// TIA Portal V17 export
// export: Created 2025-03-13T10:29:52.3164471Z, ExportSetting WithDefaults, DisplayName Totally Integrated Automation Portal, DisplayVersion V17 Update 8, DisplayName TIA Portal Openness, DisplayVersion V17 Update 8, DisplayName TIA Portal Version Control Interface, DisplayVersion V17, DisplayName SINAMICS Startdrive Advanced, DisplayVersion V17 SP2, DisplayName SINAMICS Startdrive G110M, G120, G120C, G120D, G120P, G115D, DisplayVersion V17 SP2, DisplayName SINAMICS Startdrive G130, G150, S120, S150, SINAMICS MV, S210, DisplayVersion V17 SP2, DisplayName STEP 7 Professional, DisplayVersion V17 Update 8, DisplayName SINUMERIK ONE STEP 7 Toolbox, DisplayVersion V17 Update 12, DisplayName SINUMERIK 840D sl STEP 7 Toolbox, DisplayVersion V17 Update 12, DisplayName STEP 7 Safety, DisplayVersion V17 Update 6, DisplayName WinCC Advanced, DisplayVersion V17 Update 8
FUNCTION "FC7455_QUALITY_PART_COUNTER_CLADDING" : Void   // FC7455, LAD
{ S7_Optimized_Access := 'FALSE' }
AUTHOR : ETXETAR
NAME : GM-QC
VERSION : 1.0
// stored: AutoNumber false, IsIECCheckEnabled false, SetENOAutomatically false, UDAEnableTagReadback false
   VAR_TEMP
      VALUE_0 : Real;
      AUX_FAULT : Bool;
   END_VAR
   VAR CONSTANT
      FC_NUMBER : DInt := 7455;
   END_VAR
   VAR_TEMP   // added for the SCL form of the ladder/FBD networks
      _w1 : Bool;
      _w2 : Bool;
   END_VAR
BEGIN

REGION Network 1: PART COUNTER
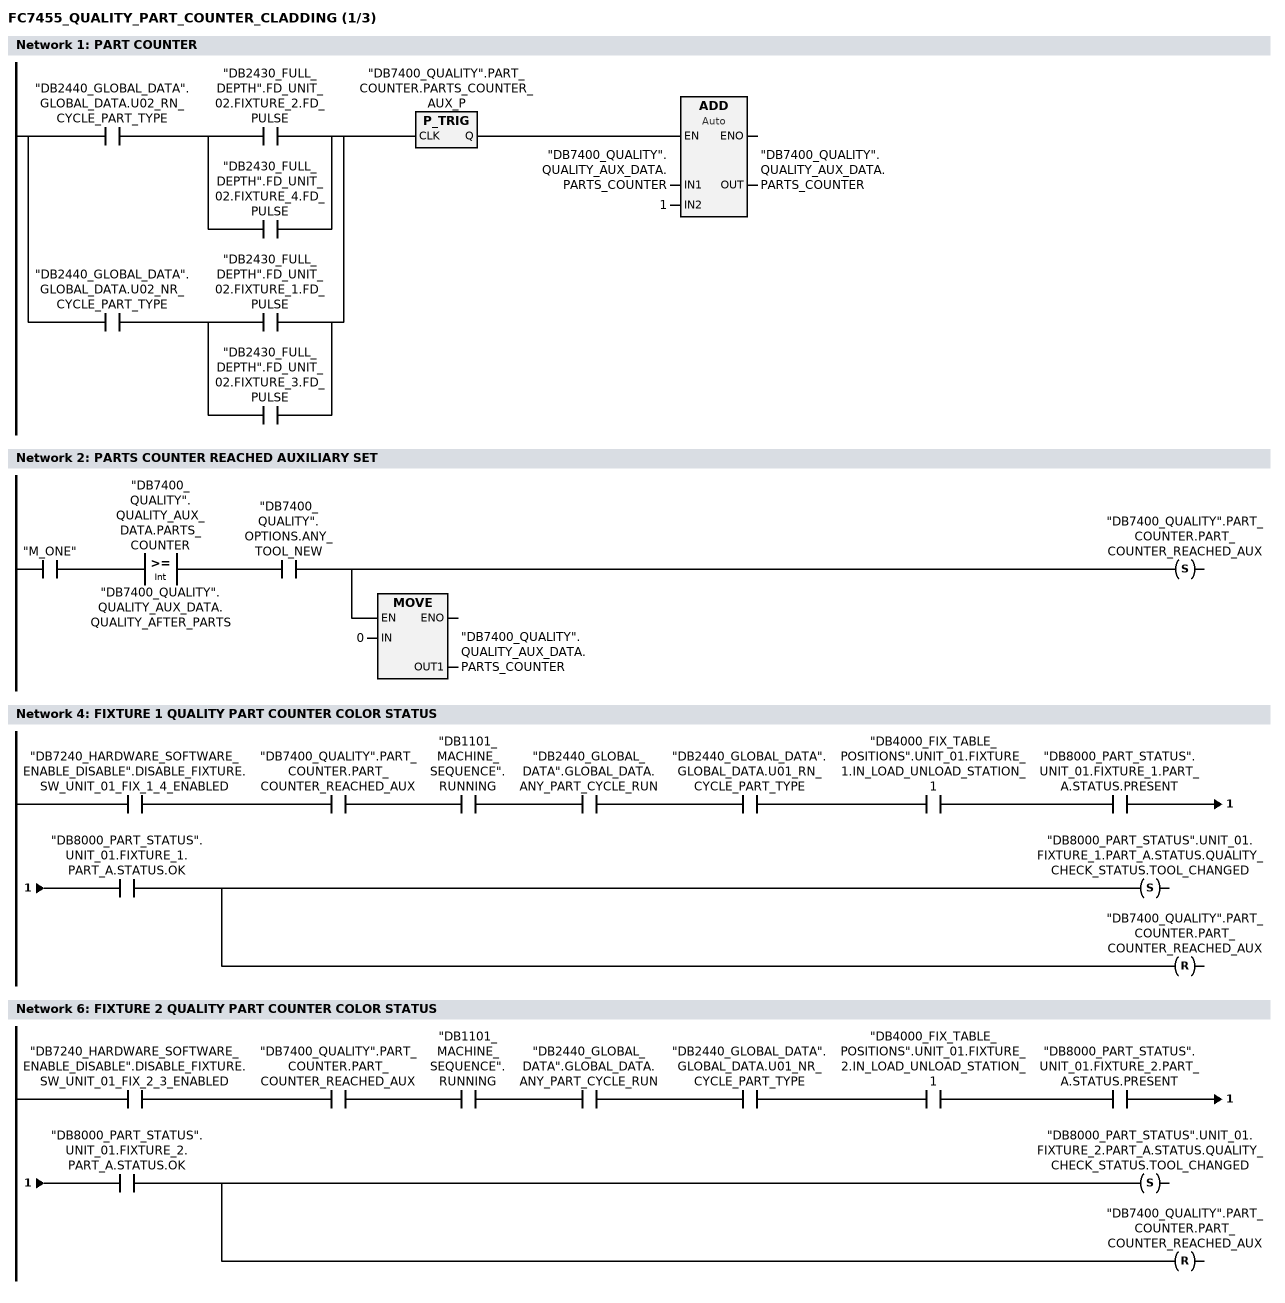
   RUNG wire#powerrail
      Contact( "DB2440_GLOBAL_DATA".GLOBAL_DATA.U02_RN_CYCLE_PART_TYPE )
      wire#w1
      Contact( "DB2430_FULL_DEPTH".FD_UNIT_02.FIXTURE_2.FD_PULSE )
      wire#w2
      P_Trig( "DB7400_QUALITY".PART_COUNTER.PARTS_COUNTER_AUX_P )
      Add(in1 := "DB7400_QUALITY".QUALITY_AUX_DATA.PARTS_COUNTER, in2 := 1, out => "DB7400_QUALITY".QUALITY_AUX_DATA.PARTS_COUNTER)
   END_RUNG
   RUNG wire#w1
      Contact( "DB2430_FULL_DEPTH".FD_UNIT_02.FIXTURE_4.FD_PULSE )
   END_RUNG wire#w2
   RUNG wire#powerrail
      Contact( "DB2440_GLOBAL_DATA".GLOBAL_DATA.U02_NR_CYCLE_PART_TYPE )
      wire#w3
      Contact( "DB2430_FULL_DEPTH".FD_UNIT_02.FIXTURE_1.FD_PULSE )
   END_RUNG wire#w2
   RUNG wire#w3
      Contact( "DB2430_FULL_DEPTH".FD_UNIT_02.FIXTURE_3.FD_PULSE )
   END_RUNG wire#w2
   // the same network as SCL:
   #_w1 := ("DB2440_GLOBAL_DATA".GLOBAL_DATA.U02_RN_CYCLE_PART_TYPE AND ("DB2430_FULL_DEPTH".FD_UNIT_02.FIXTURE_2.FD_PULSE OR "DB2430_FULL_DEPTH".FD_UNIT_02.FIXTURE_4.FD_PULSE)) OR ("DB2440_GLOBAL_DATA".GLOBAL_DATA.U02_NR_CYCLE_PART_TYPE AND ("DB2430_FULL_DEPTH".FD_UNIT_02.FIXTURE_1.FD_PULSE OR "DB2430_FULL_DEPTH".FD_UNIT_02.FIXTURE_3.FD_PULSE));
   #_w2 := #_w1 AND NOT "DB7400_QUALITY".PART_COUNTER.PARTS_COUNTER_AUX_P;   // rising edge
   "DB7400_QUALITY".PART_COUNTER.PARTS_COUNTER_AUX_P := #_w1;
   IF #_w2 THEN
       "DB7400_QUALITY".QUALITY_AUX_DATA.PARTS_COUNTER := "DB7400_QUALITY".QUALITY_AUX_DATA.PARTS_COUNTER + 1;
   END_IF;
END_REGION

REGION Network 2: PARTS COUNTER REACHED AUXILIARY SET
   RUNG wire#powerrail
      Contact( "M_ONE" )
      { S7_Templates := "SrcType := Int" } GE_Contact(in1 := "DB7400_QUALITY".QUALITY_AUX_DATA.PARTS_COUNTER, in2 := "DB7400_QUALITY".QUALITY_AUX_DATA.QUALITY_AFTER_PARTS)
      Contact( "DB7400_QUALITY".OPTIONS.ANY_TOOL_NEW )
      wire#w1
      S_Coil( "DB7400_QUALITY".PART_COUNTER.PART_COUNTER_REACHED_AUX )
   END_RUNG
   RUNG wire#w1
      Move(in := 0, out1 => "DB7400_QUALITY".QUALITY_AUX_DATA.PARTS_COUNTER)
   END_RUNG
   // the same network as SCL:
   IF "M_ONE" AND ("DB7400_QUALITY".QUALITY_AUX_DATA.PARTS_COUNTER >= "DB7400_QUALITY".QUALITY_AUX_DATA.QUALITY_AFTER_PARTS) AND "DB7400_QUALITY".OPTIONS.ANY_TOOL_NEW THEN
       "DB7400_QUALITY".PART_COUNTER.PART_COUNTER_REACHED_AUX := TRUE;
       "DB7400_QUALITY".QUALITY_AUX_DATA.PARTS_COUNTER := 0;
   END_IF;
END_REGION

REGION Network 3: /////_FIXTURE_1_/////
END_REGION

REGION Network 4: FIXTURE 1 QUALITY PART COUNTER COLOR STATUS
   RUNG wire#powerrail
      Contact( "DB7240_HARDWARE_SOFTWARE_ENABLE_DISABLE".DISABLE_FIXTURE.SW_UNIT_01_FIX_1_4_ENABLED )
      Contact( "DB7400_QUALITY".PART_COUNTER.PART_COUNTER_REACHED_AUX )
      Contact( "DB1101_MACHINE_SEQUENCE".RUNNING )
      Contact( "DB2440_GLOBAL_DATA".GLOBAL_DATA.ANY_PART_CYCLE_RUN )
      Contact( "DB2440_GLOBAL_DATA".GLOBAL_DATA.U01_RN_CYCLE_PART_TYPE )
      Contact( "DB4000_FIX_TABLE_POSITIONS".UNIT_01.FIXTURE_1.IN_LOAD_UNLOAD_STATION_1 )
      Contact( "DB8000_PART_STATUS".UNIT_01.FIXTURE_1.PART_A.STATUS.PRESENT )
      Contact( "DB8000_PART_STATUS".UNIT_01.FIXTURE_1.PART_A.STATUS.OK )
      wire#w1
      S_Coil( "DB8000_PART_STATUS".UNIT_01.FIXTURE_1.PART_A.STATUS.QUALITY_CHECK_STATUS.TOOL_CHANGED )
   END_RUNG
   RUNG wire#w1
      R_Coil( "DB7400_QUALITY".PART_COUNTER.PART_COUNTER_REACHED_AUX )
   END_RUNG
   // the same network as SCL:
   IF "DB7240_HARDWARE_SOFTWARE_ENABLE_DISABLE".DISABLE_FIXTURE.SW_UNIT_01_FIX_1_4_ENABLED AND "DB7400_QUALITY".PART_COUNTER.PART_COUNTER_REACHED_AUX AND "DB1101_MACHINE_SEQUENCE".RUNNING AND "DB2440_GLOBAL_DATA".GLOBAL_DATA.ANY_PART_CYCLE_RUN AND "DB2440_GLOBAL_DATA".GLOBAL_DATA.U01_RN_CYCLE_PART_TYPE AND "DB4000_FIX_TABLE_POSITIONS".UNIT_01.FIXTURE_1.IN_LOAD_UNLOAD_STATION_1 AND "DB8000_PART_STATUS".UNIT_01.FIXTURE_1.PART_A.STATUS.PRESENT AND "DB8000_PART_STATUS".UNIT_01.FIXTURE_1.PART_A.STATUS.OK THEN
       "DB8000_PART_STATUS".UNIT_01.FIXTURE_1.PART_A.STATUS.QUALITY_CHECK_STATUS.TOOL_CHANGED := TRUE;
       "DB7400_QUALITY".PART_COUNTER.PART_COUNTER_REACHED_AUX := FALSE;
   END_IF;
END_REGION

REGION Network 5: /////_FIXTURE_2_/////
END_REGION

REGION Network 6: FIXTURE 2 QUALITY PART COUNTER COLOR STATUS
   RUNG wire#powerrail
      Contact( "DB7240_HARDWARE_SOFTWARE_ENABLE_DISABLE".DISABLE_FIXTURE.SW_UNIT_01_FIX_2_3_ENABLED )
      Contact( "DB7400_QUALITY".PART_COUNTER.PART_COUNTER_REACHED_AUX )
      Contact( "DB1101_MACHINE_SEQUENCE".RUNNING )
      Contact( "DB2440_GLOBAL_DATA".GLOBAL_DATA.ANY_PART_CYCLE_RUN )
      Contact( "DB2440_GLOBAL_DATA".GLOBAL_DATA.U01_NR_CYCLE_PART_TYPE )
      Contact( "DB4000_FIX_TABLE_POSITIONS".UNIT_01.FIXTURE_2.IN_LOAD_UNLOAD_STATION_1 )
      Contact( "DB8000_PART_STATUS".UNIT_01.FIXTURE_2.PART_A.STATUS.PRESENT )
      Contact( "DB8000_PART_STATUS".UNIT_01.FIXTURE_2.PART_A.STATUS.OK )
      wire#w1
      S_Coil( "DB8000_PART_STATUS".UNIT_01.FIXTURE_2.PART_A.STATUS.QUALITY_CHECK_STATUS.TOOL_CHANGED )
   END_RUNG
   RUNG wire#w1
      R_Coil( "DB7400_QUALITY".PART_COUNTER.PART_COUNTER_REACHED_AUX )
   END_RUNG
   // the same network as SCL:
   IF "DB7240_HARDWARE_SOFTWARE_ENABLE_DISABLE".DISABLE_FIXTURE.SW_UNIT_01_FIX_2_3_ENABLED AND "DB7400_QUALITY".PART_COUNTER.PART_COUNTER_REACHED_AUX AND "DB1101_MACHINE_SEQUENCE".RUNNING AND "DB2440_GLOBAL_DATA".GLOBAL_DATA.ANY_PART_CYCLE_RUN AND "DB2440_GLOBAL_DATA".GLOBAL_DATA.U01_NR_CYCLE_PART_TYPE AND "DB4000_FIX_TABLE_POSITIONS".UNIT_01.FIXTURE_2.IN_LOAD_UNLOAD_STATION_1 AND "DB8000_PART_STATUS".UNIT_01.FIXTURE_2.PART_A.STATUS.PRESENT AND "DB8000_PART_STATUS".UNIT_01.FIXTURE_2.PART_A.STATUS.OK THEN
       "DB8000_PART_STATUS".UNIT_01.FIXTURE_2.PART_A.STATUS.QUALITY_CHECK_STATUS.TOOL_CHANGED := TRUE;
       "DB7400_QUALITY".PART_COUNTER.PART_COUNTER_REACHED_AUX := FALSE;
   END_IF;
END_REGION

REGION Network 7: /////_FIXTURE_3_/////
END_REGION

REGION Network 8: FIXTURE 3 QUALITY PART COUNTER COLOR STATUS
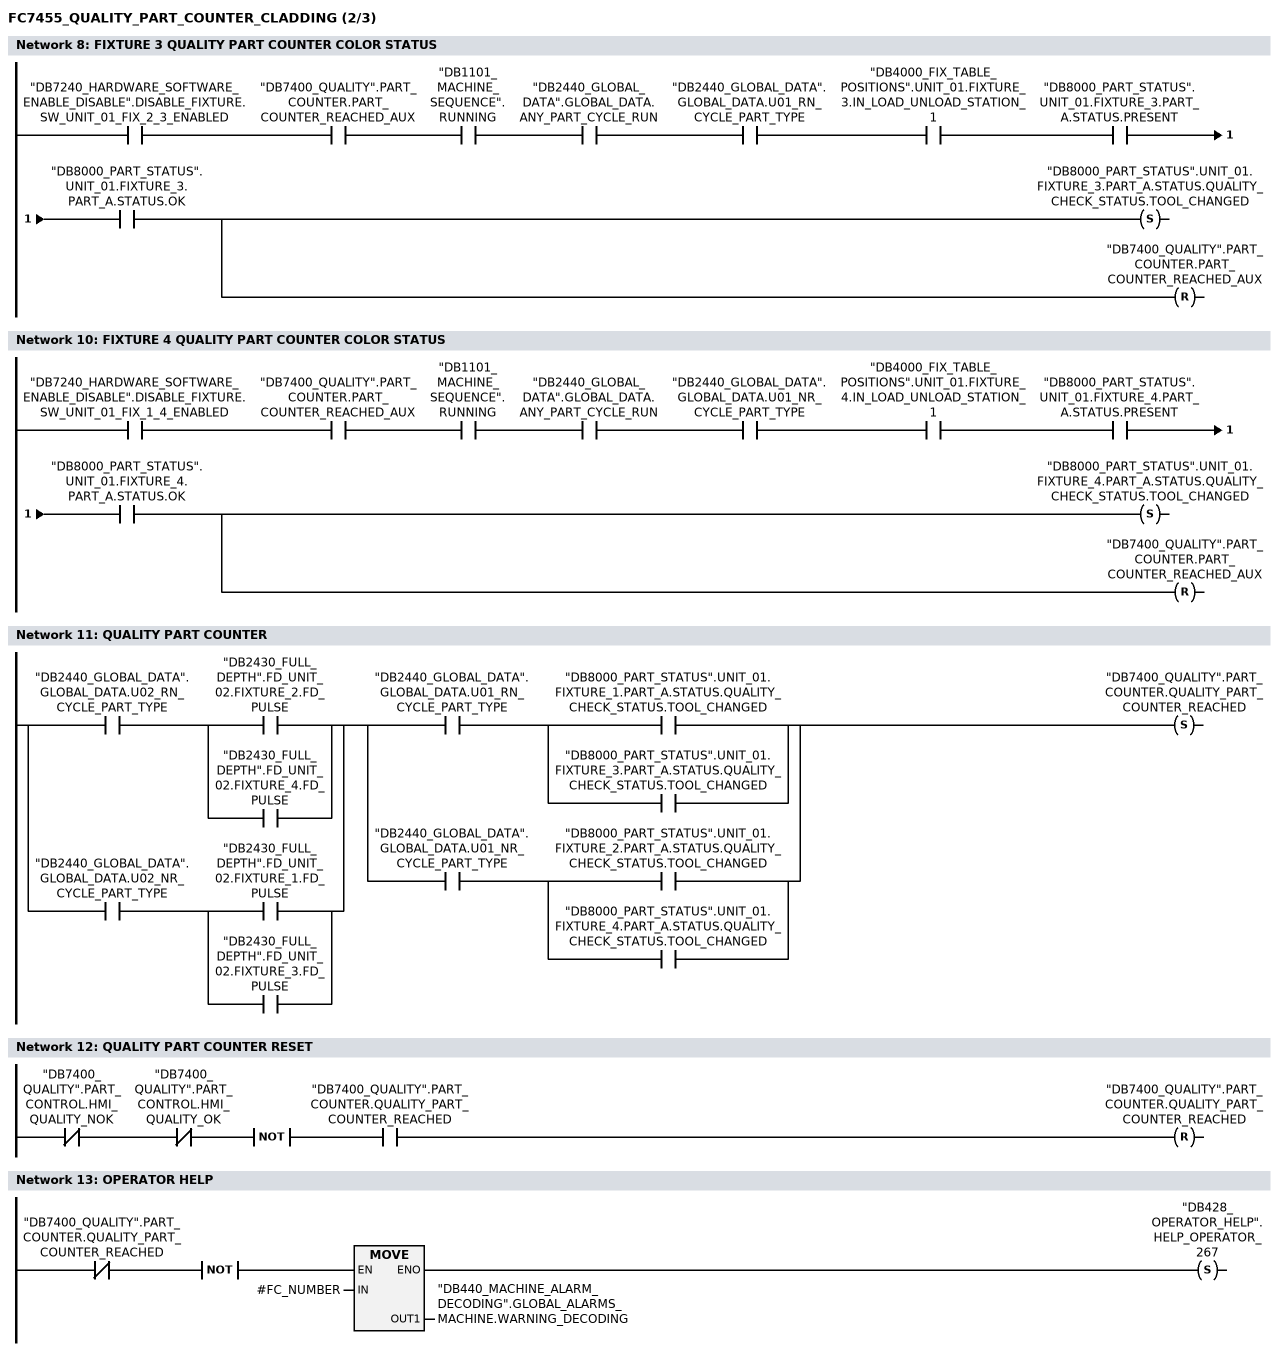
   RUNG wire#powerrail
      Contact( "DB7240_HARDWARE_SOFTWARE_ENABLE_DISABLE".DISABLE_FIXTURE.SW_UNIT_01_FIX_2_3_ENABLED )
      Contact( "DB7400_QUALITY".PART_COUNTER.PART_COUNTER_REACHED_AUX )
      Contact( "DB1101_MACHINE_SEQUENCE".RUNNING )
      Contact( "DB2440_GLOBAL_DATA".GLOBAL_DATA.ANY_PART_CYCLE_RUN )
      Contact( "DB2440_GLOBAL_DATA".GLOBAL_DATA.U01_RN_CYCLE_PART_TYPE )
      Contact( "DB4000_FIX_TABLE_POSITIONS".UNIT_01.FIXTURE_3.IN_LOAD_UNLOAD_STATION_1 )
      Contact( "DB8000_PART_STATUS".UNIT_01.FIXTURE_3.PART_A.STATUS.PRESENT )
      Contact( "DB8000_PART_STATUS".UNIT_01.FIXTURE_3.PART_A.STATUS.OK )
      wire#w1
      S_Coil( "DB8000_PART_STATUS".UNIT_01.FIXTURE_3.PART_A.STATUS.QUALITY_CHECK_STATUS.TOOL_CHANGED )
   END_RUNG
   RUNG wire#w1
      R_Coil( "DB7400_QUALITY".PART_COUNTER.PART_COUNTER_REACHED_AUX )
   END_RUNG
   // the same network as SCL:
   IF "DB7240_HARDWARE_SOFTWARE_ENABLE_DISABLE".DISABLE_FIXTURE.SW_UNIT_01_FIX_2_3_ENABLED AND "DB7400_QUALITY".PART_COUNTER.PART_COUNTER_REACHED_AUX AND "DB1101_MACHINE_SEQUENCE".RUNNING AND "DB2440_GLOBAL_DATA".GLOBAL_DATA.ANY_PART_CYCLE_RUN AND "DB2440_GLOBAL_DATA".GLOBAL_DATA.U01_RN_CYCLE_PART_TYPE AND "DB4000_FIX_TABLE_POSITIONS".UNIT_01.FIXTURE_3.IN_LOAD_UNLOAD_STATION_1 AND "DB8000_PART_STATUS".UNIT_01.FIXTURE_3.PART_A.STATUS.PRESENT AND "DB8000_PART_STATUS".UNIT_01.FIXTURE_3.PART_A.STATUS.OK THEN
       "DB8000_PART_STATUS".UNIT_01.FIXTURE_3.PART_A.STATUS.QUALITY_CHECK_STATUS.TOOL_CHANGED := TRUE;
       "DB7400_QUALITY".PART_COUNTER.PART_COUNTER_REACHED_AUX := FALSE;
   END_IF;
END_REGION

REGION Network 9: /////_FIXTURE_4_/////
END_REGION

REGION Network 10: FIXTURE 4 QUALITY PART COUNTER COLOR STATUS
   RUNG wire#powerrail
      Contact( "DB7240_HARDWARE_SOFTWARE_ENABLE_DISABLE".DISABLE_FIXTURE.SW_UNIT_01_FIX_1_4_ENABLED )
      Contact( "DB7400_QUALITY".PART_COUNTER.PART_COUNTER_REACHED_AUX )
      Contact( "DB1101_MACHINE_SEQUENCE".RUNNING )
      Contact( "DB2440_GLOBAL_DATA".GLOBAL_DATA.ANY_PART_CYCLE_RUN )
      Contact( "DB2440_GLOBAL_DATA".GLOBAL_DATA.U01_NR_CYCLE_PART_TYPE )
      Contact( "DB4000_FIX_TABLE_POSITIONS".UNIT_01.FIXTURE_4.IN_LOAD_UNLOAD_STATION_1 )
      Contact( "DB8000_PART_STATUS".UNIT_01.FIXTURE_4.PART_A.STATUS.PRESENT )
      Contact( "DB8000_PART_STATUS".UNIT_01.FIXTURE_4.PART_A.STATUS.OK )
      wire#w1
      S_Coil( "DB8000_PART_STATUS".UNIT_01.FIXTURE_4.PART_A.STATUS.QUALITY_CHECK_STATUS.TOOL_CHANGED )
   END_RUNG
   RUNG wire#w1
      R_Coil( "DB7400_QUALITY".PART_COUNTER.PART_COUNTER_REACHED_AUX )
   END_RUNG
   // the same network as SCL:
   IF "DB7240_HARDWARE_SOFTWARE_ENABLE_DISABLE".DISABLE_FIXTURE.SW_UNIT_01_FIX_1_4_ENABLED AND "DB7400_QUALITY".PART_COUNTER.PART_COUNTER_REACHED_AUX AND "DB1101_MACHINE_SEQUENCE".RUNNING AND "DB2440_GLOBAL_DATA".GLOBAL_DATA.ANY_PART_CYCLE_RUN AND "DB2440_GLOBAL_DATA".GLOBAL_DATA.U01_NR_CYCLE_PART_TYPE AND "DB4000_FIX_TABLE_POSITIONS".UNIT_01.FIXTURE_4.IN_LOAD_UNLOAD_STATION_1 AND "DB8000_PART_STATUS".UNIT_01.FIXTURE_4.PART_A.STATUS.PRESENT AND "DB8000_PART_STATUS".UNIT_01.FIXTURE_4.PART_A.STATUS.OK THEN
       "DB8000_PART_STATUS".UNIT_01.FIXTURE_4.PART_A.STATUS.QUALITY_CHECK_STATUS.TOOL_CHANGED := TRUE;
       "DB7400_QUALITY".PART_COUNTER.PART_COUNTER_REACHED_AUX := FALSE;
   END_IF;
END_REGION

REGION Network 11: QUALITY PART COUNTER
   RUNG wire#powerrail
      Contact( "DB2440_GLOBAL_DATA".GLOBAL_DATA.U02_RN_CYCLE_PART_TYPE )
      wire#w1
      Contact( "DB2430_FULL_DEPTH".FD_UNIT_02.FIXTURE_2.FD_PULSE )
      wire#w2
      Contact( "DB2440_GLOBAL_DATA".GLOBAL_DATA.U01_RN_CYCLE_PART_TYPE )
      wire#w4
      Contact( "DB8000_PART_STATUS".UNIT_01.FIXTURE_1.PART_A.STATUS.QUALITY_CHECK_STATUS.TOOL_CHANGED )
      wire#w5
      S_Coil( "DB7400_QUALITY".PART_COUNTER.QUALITY_PART_COUNTER_REACHED )
   END_RUNG
   RUNG wire#w1
      Contact( "DB2430_FULL_DEPTH".FD_UNIT_02.FIXTURE_4.FD_PULSE )
   END_RUNG wire#w2
   RUNG wire#powerrail
      Contact( "DB2440_GLOBAL_DATA".GLOBAL_DATA.U02_NR_CYCLE_PART_TYPE )
      wire#w3
      Contact( "DB2430_FULL_DEPTH".FD_UNIT_02.FIXTURE_1.FD_PULSE )
   END_RUNG wire#w2
   RUNG wire#w3
      Contact( "DB2430_FULL_DEPTH".FD_UNIT_02.FIXTURE_3.FD_PULSE )
   END_RUNG wire#w2
   RUNG wire#w4
      Contact( "DB8000_PART_STATUS".UNIT_01.FIXTURE_3.PART_A.STATUS.QUALITY_CHECK_STATUS.TOOL_CHANGED )
   END_RUNG wire#w5
   RUNG wire#w2
      Contact( "DB2440_GLOBAL_DATA".GLOBAL_DATA.U01_NR_CYCLE_PART_TYPE )
      wire#w6
      Contact( "DB8000_PART_STATUS".UNIT_01.FIXTURE_2.PART_A.STATUS.QUALITY_CHECK_STATUS.TOOL_CHANGED )
   END_RUNG wire#w5
   RUNG wire#w6
      Contact( "DB8000_PART_STATUS".UNIT_01.FIXTURE_4.PART_A.STATUS.QUALITY_CHECK_STATUS.TOOL_CHANGED )
   END_RUNG wire#w5
   // the same network as SCL:
   IF (("DB2440_GLOBAL_DATA".GLOBAL_DATA.U02_RN_CYCLE_PART_TYPE AND ("DB2430_FULL_DEPTH".FD_UNIT_02.FIXTURE_2.FD_PULSE OR "DB2430_FULL_DEPTH".FD_UNIT_02.FIXTURE_4.FD_PULSE)) OR ("DB2440_GLOBAL_DATA".GLOBAL_DATA.U02_NR_CYCLE_PART_TYPE AND ("DB2430_FULL_DEPTH".FD_UNIT_02.FIXTURE_1.FD_PULSE OR "DB2430_FULL_DEPTH".FD_UNIT_02.FIXTURE_3.FD_PULSE))) AND (("DB2440_GLOBAL_DATA".GLOBAL_DATA.U01_RN_CYCLE_PART_TYPE AND ("DB8000_PART_STATUS".UNIT_01.FIXTURE_1.PART_A.STATUS.QUALITY_CHECK_STATUS.TOOL_CHANGED OR "DB8000_PART_STATUS".UNIT_01.FIXTURE_3.PART_A.STATUS.QUALITY_CHECK_STATUS.TOOL_CHANGED)) OR ("DB2440_GLOBAL_DATA".GLOBAL_DATA.U01_NR_CYCLE_PART_TYPE AND ("DB8000_PART_STATUS".UNIT_01.FIXTURE_2.PART_A.STATUS.QUALITY_CHECK_STATUS.TOOL_CHANGED OR "DB8000_PART_STATUS".UNIT_01.FIXTURE_4.PART_A.STATUS.QUALITY_CHECK_STATUS.TOOL_CHANGED))) THEN
       "DB7400_QUALITY".PART_COUNTER.QUALITY_PART_COUNTER_REACHED := TRUE;
   END_IF;
END_REGION

REGION Network 12: QUALITY PART COUNTER RESET
   RUNG wire#powerrail
      I_Contact( "DB7400_QUALITY".PART_CONTROL.HMI_QUALITY_NOK )
      I_Contact( "DB7400_QUALITY".PART_CONTROL.HMI_QUALITY_OK )
      Not()
      Contact( "DB7400_QUALITY".PART_COUNTER.QUALITY_PART_COUNTER_REACHED )
      R_Coil( "DB7400_QUALITY".PART_COUNTER.QUALITY_PART_COUNTER_REACHED )
   END_RUNG
   // the same network as SCL:
   IF NOT (NOT "DB7400_QUALITY".PART_CONTROL.HMI_QUALITY_NOK AND NOT "DB7400_QUALITY".PART_CONTROL.HMI_QUALITY_OK) AND "DB7400_QUALITY".PART_COUNTER.QUALITY_PART_COUNTER_REACHED THEN
       "DB7400_QUALITY".PART_COUNTER.QUALITY_PART_COUNTER_REACHED := FALSE;
   END_IF;
END_REGION

REGION Network 13: OPERATOR HELP
   RUNG wire#powerrail
      I_Contact( "DB7400_QUALITY".PART_COUNTER.QUALITY_PART_COUNTER_REACHED )
      Not()
      { S7_GenerateENO := "TRUE" } Move(in := #FC_NUMBER, out1 => "DB440_MACHINE_ALARM_DECODING".GLOBAL_ALARMS_MACHINE.WARNING_DECODING)
      S_Coil( "DB428_OPERATOR_HELP".HELP_OPERATOR_267 )
   END_RUNG
   // the same network as SCL:
   // ENO of a box is taken as its EN; it also drops when the box reports an error
   IF NOT (NOT "DB7400_QUALITY".PART_COUNTER.QUALITY_PART_COUNTER_REACHED) THEN
       "DB440_MACHINE_ALARM_DECODING".GLOBAL_ALARMS_MACHINE.WARNING_DECODING := #FC_NUMBER;
       "DB428_OPERATOR_HELP".HELP_OPERATOR_267 := TRUE;
   END_IF;
END_REGION

REGION Network 14: (WRN) QUALITY PART INSPECTION AFTER PART COUNTER REACHED
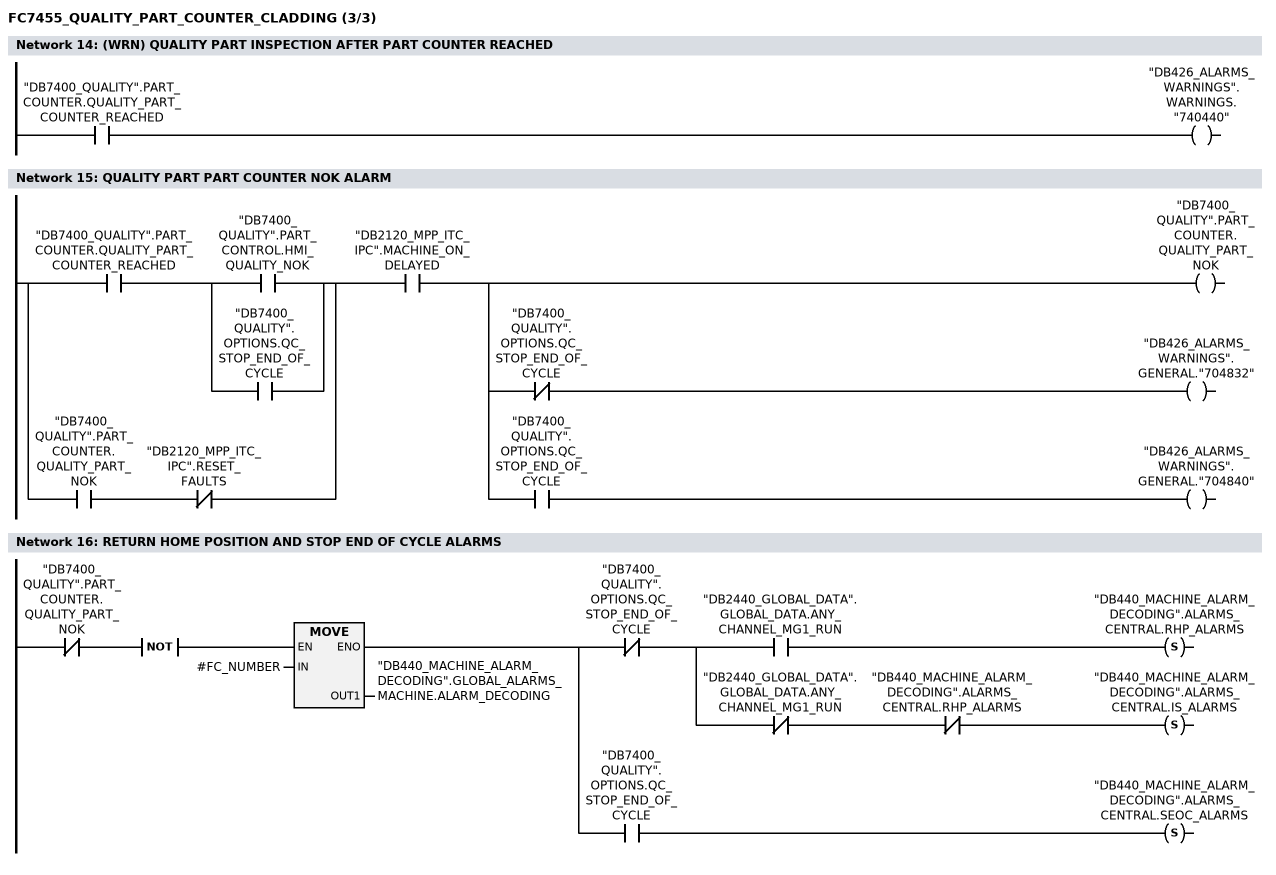
   RUNG wire#powerrail
      Contact( "DB7400_QUALITY".PART_COUNTER.QUALITY_PART_COUNTER_REACHED )
      Coil( "DB426_ALARMS_WARNINGS".WARNINGS."740440" )
   END_RUNG
   // the same network as SCL:
   "DB426_ALARMS_WARNINGS".WARNINGS."740440" := "DB7400_QUALITY".PART_COUNTER.QUALITY_PART_COUNTER_REACHED;
END_REGION

REGION Network 15: QUALITY PART PART COUNTER NOK ALARM
   RUNG wire#powerrail
      Contact( "DB7400_QUALITY".PART_COUNTER.QUALITY_PART_COUNTER_REACHED )
      wire#w1
      Contact( "DB7400_QUALITY".PART_CONTROL.HMI_QUALITY_NOK )
      wire#w2
      Contact( "DB2120_MPP_ITC_IPC".MACHINE_ON_DELAYED )
      wire#w3
      Coil( "DB7400_QUALITY".PART_COUNTER.QUALITY_PART_NOK )
   END_RUNG
   RUNG wire#w1
      Contact( "DB7400_QUALITY".OPTIONS.QC_STOP_END_OF_CYCLE )
   END_RUNG wire#w2
   RUNG wire#powerrail
      Contact( "DB7400_QUALITY".PART_COUNTER.QUALITY_PART_NOK )
      I_Contact( "DB2120_MPP_ITC_IPC".RESET_FAULTS )
   END_RUNG wire#w2
   RUNG wire#w3
      I_Contact( "DB7400_QUALITY".OPTIONS.QC_STOP_END_OF_CYCLE )
      Coil( "DB426_ALARMS_WARNINGS".GENERAL."704832" )
   END_RUNG
   RUNG wire#w3
      Contact( "DB7400_QUALITY".OPTIONS.QC_STOP_END_OF_CYCLE )
      Coil( "DB426_ALARMS_WARNINGS".GENERAL."704840" )
   END_RUNG
   // the same network as SCL:
   "DB7400_QUALITY".PART_COUNTER.QUALITY_PART_NOK := (("DB7400_QUALITY".PART_COUNTER.QUALITY_PART_COUNTER_REACHED AND ("DB7400_QUALITY".PART_CONTROL.HMI_QUALITY_NOK OR "DB7400_QUALITY".OPTIONS.QC_STOP_END_OF_CYCLE)) OR ("DB7400_QUALITY".PART_COUNTER.QUALITY_PART_NOK AND NOT "DB2120_MPP_ITC_IPC".RESET_FAULTS)) AND "DB2120_MPP_ITC_IPC".MACHINE_ON_DELAYED;
   "DB426_ALARMS_WARNINGS".GENERAL."704832" := "DB7400_QUALITY".PART_COUNTER.QUALITY_PART_NOK AND NOT "DB7400_QUALITY".OPTIONS.QC_STOP_END_OF_CYCLE;
   "DB426_ALARMS_WARNINGS".GENERAL."704840" := "DB7400_QUALITY".PART_COUNTER.QUALITY_PART_NOK AND "DB7400_QUALITY".OPTIONS.QC_STOP_END_OF_CYCLE;
END_REGION

REGION Network 16: RETURN HOME POSITION AND STOP END OF CYCLE ALARMS
   RUNG wire#powerrail
      I_Contact( "DB7400_QUALITY".PART_COUNTER.QUALITY_PART_NOK )
      Not()
      { S7_GenerateENO := "TRUE" } Move(in := #FC_NUMBER, out1 => "DB440_MACHINE_ALARM_DECODING".GLOBAL_ALARMS_MACHINE.ALARM_DECODING)
      wire#w1
      I_Contact( "DB7400_QUALITY".OPTIONS.QC_STOP_END_OF_CYCLE )
      wire#w2
      Contact( "DB2440_GLOBAL_DATA".GLOBAL_DATA.ANY_CHANNEL_MG1_RUN )
      S_Coil( "DB440_MACHINE_ALARM_DECODING".ALARMS_CENTRAL.RHP_ALARMS )
   END_RUNG
   RUNG wire#w2
      I_Contact( "DB2440_GLOBAL_DATA".GLOBAL_DATA.ANY_CHANNEL_MG1_RUN )
      I_Contact( "DB440_MACHINE_ALARM_DECODING".ALARMS_CENTRAL.RHP_ALARMS )
      S_Coil( "DB440_MACHINE_ALARM_DECODING".ALARMS_CENTRAL.IS_ALARMS )
   END_RUNG
   RUNG wire#w1
      Contact( "DB7400_QUALITY".OPTIONS.QC_STOP_END_OF_CYCLE )
      S_Coil( "DB440_MACHINE_ALARM_DECODING".ALARMS_CENTRAL.SEOC_ALARMS )
   END_RUNG
   // the same network as SCL:
   // ENO of a box is taken as its EN; it also drops when the box reports an error
   #_w1 := NOT (NOT "DB7400_QUALITY".PART_COUNTER.QUALITY_PART_NOK);
   IF #_w1 THEN "DB440_MACHINE_ALARM_DECODING".GLOBAL_ALARMS_MACHINE.ALARM_DECODING := #FC_NUMBER; END_IF;
   #_w2 := #_w1 AND NOT "DB7400_QUALITY".OPTIONS.QC_STOP_END_OF_CYCLE;
   IF #_w2 AND "DB2440_GLOBAL_DATA".GLOBAL_DATA.ANY_CHANNEL_MG1_RUN THEN
       "DB440_MACHINE_ALARM_DECODING".ALARMS_CENTRAL.RHP_ALARMS := TRUE;
   END_IF;
   IF #_w2 AND NOT "DB2440_GLOBAL_DATA".GLOBAL_DATA.ANY_CHANNEL_MG1_RUN AND NOT "DB440_MACHINE_ALARM_DECODING".ALARMS_CENTRAL.RHP_ALARMS THEN
       "DB440_MACHINE_ALARM_DECODING".ALARMS_CENTRAL.IS_ALARMS := TRUE;
   END_IF;
   IF #_w1 AND "DB7400_QUALITY".OPTIONS.QC_STOP_END_OF_CYCLE THEN
       "DB440_MACHINE_ALARM_DECODING".ALARMS_CENTRAL.SEOC_ALARMS := TRUE;
   END_IF;
END_REGION
END_FUNCTION
